Fanuc KAREL source: kt00532.KL

-- PROVISIONAL review KL for V940-1; original PC SHA256 35d8db5103a30de757a35d0dbcf870526a60c127a75141c7e5beaa3f736e0617
-- Incomplete behavior may be omitted. Consult companion uncertainty JSON. Do not deploy.
PROGRAM KT00532
%NOLOCKGROUP
-- UNRESOLVED_DECL P1 type=000106
-- UNRESOLVED_DECL P2 type=000199
-- UNRESOLVED_DECL OUT type=000199
BEGIN
  -- V9_ZERO_TABLE_METADATA_HINT layout=0001; no indexed target words; source/name/runtime held
  -- UNRESOLVED_PC offsets 5-20; opcodes 2E,22,32,35
  -- UNRESOLVED_PC offsets 25-64; opcodes 49,7E,49,7E,60,7E,4A
  -- UNRESOLVED_PC offsets 69-73; opcodes 7F
END KT00532
